TYPE E_AxisMotionState :
(
	Init := 10,
	MoveEnabled := 3000,
	Error := 9000
);
END_TYPE

(* stored: Version 1.1.0.1, ProductVersion 3.1.4018.5
   DUT E_AxisMotionState: Id {76fd406e-4c8d-41a4-9b2d-13dbdd19a9ab} *)
